FUNCTION_BLOCK ASR_2AE_TO_SR (* Composite FB for convert 2 AE to ASR *)
  (* Standard: 61499-2; Description: Copyright (c) 2026 HR Agrartechnik GmbH This program and the accompanying materials are made available under the terms of the Eclipse Public License 2.0 which is available at https://www.eclipse.org/legal/epl-2.0/ SPDX-License-Identifier: EPL-2.0 *)
  (* Version 1.0, 2026-09-06, Franz Höpfinger, HR Agrartechnik GmbH *)
  PACKAGE adapter::conversion::unidirectional;
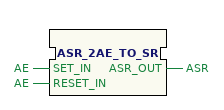
  SOCKETS
    SET_IN : adapter::types::unidirectional::AE; (* Set / Switch on *)
    RESET_IN : adapter::types::unidirectional::AE; (* Reset / Switch off *)
  END_SOCKETS
  PLUGS
    ASR_OUT : adapter::types::unidirectional::ASR; (* Adapter Output *)
  END_PLUGS
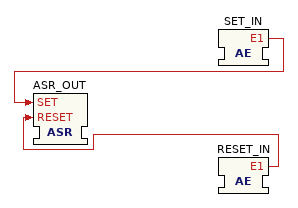
  EVENT_CONNECTIONS
    SET_IN.E1 TO ASR_OUT.SET;
    RESET_IN.E1 TO ASR_OUT.RESET;
  END_CONNECTIONS
END_FUNCTION_BLOCK
